# B&R Automation Studio project TD52 (part 21)

#### resetCyclic.st
```iecst
(*******************************************************************************
reset			general reset alarms
				definition remote reset capability for each individual alarm (according TI 1100-0111)

This code is confidential and proprietary to the INNIO Company.
It may not be used in any form, or reproduced in any manner,
without written permission of the INNIO Company.
Copyright, INNIO Company, 2023

Customized modifications: -
------------------------

History:
-------
V0.1	19-06-2009	Brindlinger, new
V3.10.0	12.01.2010	lettenb.	corr.for version 3.10.0
		15.02.2010	lettenb.	DO_W_QUITT, DO_A_QUITT added from task: pb8
		02.03.2010	lettenb.	extended remote reset command with T_FQUITT (was M_FQUITT)
								(needed for reset exhaust temp.alarms generated from task: exhaust)
V3.20.0	24.03.2010	lettenb.	amm numbers br9 (2201-2300) added
		21.05.2010				reset_alarm[1022,1056]: QUITT2_RUHE added
		27.05.2010				AMM test mode added, dianeblau software parts removed
		14.10.2010				NumAmmTest limited, loops reduced to 3999
V3.99.0	06.03.2013	lettenb.	adaption for pilot engine 6
								AB2MM.bResetRiskClass. added
V4.00.0 04.06.2014	lettenb.	write on VIS2MM.iNumAlarmTest removed(asynchr.running VIS do not change input field value!)
								(in case of illegal alarm nr.: alarm nr will NOT be changed, timer will NOT be started/=diff.to XT3)
		17.06.2014	lettenb.	iNumAlarmTestRun: set to 0 after alarmtest
V4.00.1 04.06.2014	lettenb.	bRemResMem: logic corr., rem.reset counter(5 resets)
V4.00.2 16.02.2015				warm-/cold restart message generation moved to MsgAB
V4.03.0 16.02.2015				protection test (gridcode III) schutzprüfung added
V4.04.0 03.11.2016				IN_AB.bResetRemBus added, prepared for future(wasserer-rosenheim)
		16.11.2016				bResetTrip: xTP_RemResCmd.Q removed, bugfix(reset all risk classes)
V4.05.1 07.03.2018	lettenb.	xR_TRIG_Run: bRun -> IN_AB.tPB2MM.bSys_Run, to avoid 1056 at PLC startup, bugfix
		21.03.2018				protection test mode: passlevel 30->15, request thaler
V4.07.1	24.06.2019	Schmid		valid alarm number space for alarm test/bypass increased from 3999 to 9999
V4.08.0	24.10.2019	Schmid		test bit for dry test bench added
V4.13.0	04.12.2023	Bencze		Risk Class 10 for remote reset of safety trips
		13.12.2023	Perktold	added A2374 as safety trip without remote reset
V4.14.0	16.12.2024	Maran		bugfix: reset of temporary alarm bypass when the Service button is switched off from HMI (issue #1621)

Instructions for use:
--------------------

Outstandings:
------------
*******************************************************************************)
PROGRAM _CYCLIC

	(*-----------------------------------------------------------------------------------------*)
	bResetLocVis			:=	VIS2MM.bResetLocVis;			(* local  reset from VIS  *)(* vis-button: 0>1 in moment of button release! *)
	bResetRemVis			:=	VIS2MM.bResetRemVis;			(* remote reset from VIS  *)(* vis-button: 0>1 in moment of button release! *)
	xF_TRIG_ResetRemExt(CLK	:=  IN_AB.tResetRemoteExt.Di		(* remote reset from DI   *)(* falling trigger according TÜV requirement *)
						    OR  IN_AB.bResetRemBus);			(* remote reset from fieldbus *)
	bResetRemExt			:=	xF_TRIG_ResetRemExt.Q;			(* falling trigger according TÜV requirement *)

	IF VIS2MM.bResetLocVis THEN VIS2MM.bResetLocVis := FALSE; END_IF;	(* reset vis data point  *)
	IF VIS2MM.bResetRemVis THEN VIS2MM.bResetRemVis := FALSE; END_IF;	(* reset vis data point *)

	(*-----------------------------------------------------------------------------------------*)
	QUITT		:=	bResetLocVis;								(* local  reset from VIS  *)
	VIS_FQUITT	:=	bResetRemVis;								(* remote reset from VIS *)
	E_FQUITT	:=	bResetRemExt;								(* remote reset from DI  *)

	(* remote reset ---------------------------------------------------------------------------*)
	bRemResIn	:= (E_FQUITT 	AND Para.bResetRemActive)		(* remote reset from DI  *)
				OR (VIS_FQUITT	AND Para.bResetRemActive);		(* remote reset from VIS *)

	(********************************************************************************************************************
	Safety-related application software source code (EN 13849-1 / 4.6.3): BEGIN
	*********************************************************************************************************************)

	(* If one of these alarms is ON, Remote Reset is deactivated *)
	IF OUT_AB.iMsg[1017]>0 OR		(* A1017 oil pressure low *)
		OUT_AB.iMsg[1019]>0 OR		(* A1019 engine cooling water pressure low *)
		OUT_AB.iMsg[1022]>0 OR		(* A1022 overspeed (relay) *)
		OUT_AB.iMsg[1026]>0 OR		(* A1026 shutdown failure *)
		OUT_AB.iMsg[1038]>0 OR		(* A1038 Generator reverse power *)
		OUT_AB.iMsg[1047]>0 OR		(* A1047: Misfiring failure *)
		(xEngType.Type6 AND OUT_AB.iMsg[1048]>0) OR		(* A1048 Knocking failure KLS90 *)
		OUT_AB.iMsg[1092]>0 OR		(* A1092 exhaust gas scavenging valve failure *)
		OUT_AB.iMsg[1131]>0 OR		(*  prepared spare - risk class 10 and this is only for trips 1,2 or 3. Remote reset is deactivated *)
		OUT_AB.iMsg[2295]>0 OR		(* A2295 engine room ventilation failure inlet air *)
		OUT_AB.iMsg[2296]>0 OR		(* A2296 engine room ventilation failure outlet air *)
		OUT_AB.iMsg[2315]>0 OR		(* A2315 air temperature before exhaust gas scavening valve maximum *)
		OUT_AB.iMsg[2337]>0 OR		(* A2337 temperature high exhaust gas pressure relief valve 1 *)
		OUT_AB.iMsg[2338]>0 OR		(* A2338 temperature high exhaust gas pressure relief valve 2 *)
		OUT_AB.iMsg[2374]>0	OR		(* A2374 Bursting disc triggered *)
		OUT_AB.iMsg[3330]>0 OR 		(* A3330 SAFI hardware failure *)
		OUT_AB.iMsg[3336]>0	OR		(* A3336 SAFI trigger signal missing *)
		OUT_AB.iMsg[3337]>0 OR		(* A3337 SAFI CAM / RESET pickup signal missing *)
		(xEngType.Type6 AND OUT_AB.iMsg[3339]>0) OR		(* A3339 Knocking failure *)
		(xEngType.Type6 AND OUT_AB.iMsg[3342]>0) OR		(* A3342 Knock sensor measuring sensor failure *)
		OUT_AB.iMsg[3343]>0 OR		(* A3343 ignition hardware failure *)
		OUT_AB.iMsg[3366]>0			(* A3366 exhaust gas scavenging fan failure *)
	THEN
		bRemResIn := FALSE;
                bRemResWarning := TRUE;
	END_IF;

	(********************************************************************************************************************
	Safety-related application software source code (EN 13849-1 / 4.6.3): END
	*********************************************************************************************************************)

	bRemResMem	:=	bRemResIn									(* remote reset memory,  unlock after: *)
				OR (bRemResMem 	AND NOT ton_FQ_timeout.Q		(* 6 h             					or *)
								AND NOT ton_oper.Q 				(* 1 h operation with closed GCB 	or *)
								AND(NOT bResetWarning OR bOMSS_MAT));(* local reset					       *)

	ton_oper(IN:= bRemResMem AND IN_AB.tGCB_On.Di AND IN_AB.tEng_Run.Do, PT:= T#1h);	(* reset after 1h load operation *)
	ton_FQ_timeout(IN:= bRemResMem, PT:=T#6h);											(* reset after 6h *)

	xR_TRIG_CD(CLK:=     bRemResIn);
	xR_TRIG_LD(CLK:= NOT bRemResMem);

	xTP_RemResCmd(IN:=  bRemResIn AND NOT xCTD_RRC.Q, PT:= T#1s);
	bRemResCmd := xTP_RemResCmd.Q;								(* remote reset command *)

	xCTD_RRC(CD:= xR_TRIG_CD.Q, LOAD:= xR_TRIG_LD.Q, PV:= 5);	(* count 5 avail.remote reset commands within 6h *)

	IF xCTD_RRC.CV=0 THEN	bRemResWarning := TRUE;				(* reached the available 5 remote reset within 1h/6h *)
	END_IF;
	(* if remote reset risk class lower than 0, the risk level is limited to 0 *)
	(* if remote reset risk class higher than 4, the risk level is limited to 4 *)
	IF Para.iResetRemRiskClass < 0 THEN Para.iResetRemRiskClass := 0;
	ELSIF Para.iResetRemRiskClass > 4 THEN Para.iResetRemRiskClass := 4;
	END_IF;

	(*-----------------------------------------------------------------------------------------*)
	xTP_Reset(IN:= QUITT OR E_QUITT, PT:= T#100ms);
	IF bDryTB_AB THEN
		xTP_DryTB_AB(IN:= bDryTB_AB, PT:= T#8h);
	ELSE
		xTP_DryTB_AB(IN:= FALSE, PT:= T#0s);
	END_IF;

	bResetWarning	:=	xTP_Reset.Q;
	bResetTrip		:=	bResetWarning AND (NOT bOMSS_MAT OR xTP_DryTB_AB.Q);

	(* remote reset commands *)
	CASE Para.iResetRemRiskClass OF
		0:	bResetRiskClass0 :=	bRemResCmd;
		1:	bResetRiskClass1 :=	bRemResCmd;
		2:	bResetRiskClass2 :=	bRemResCmd;
		3:	bResetRiskClass3 :=	bRemResCmd;
		4:	bResetRiskClass4 :=	bRemResCmd;
	END_CASE;

	(*-----------------------------------------------------------------------------------------*)
	(* monitoring on pulse (safety loop) *)
                                                        (* falling trigger according TÜV requirement *)
	xR_TRIG_Run(CLK:= IN_AB.tPB2MM.bSys_Run);			(* EN ISO 13849-1 / 5.2.2, = reset after push button release) *)
	xTP_MonOn(IN:= (xR_TRIG_Run.Q AND     IN_AB.tGCB_RUC.Do)
			    OR (QUITT         AND NOT IN_AB.tSafetyLoop_Eng.Di AND NOT bN_EngStart AND (NOT bOMSS_MAT OR xTP_DryTB_AB.Q)), PT:= T#1s);

	OUT_AB.tMonitoringOn.Do := xTP_MonOn.Q;				(* ex UW_EIN *)

	f_trig_UW_EIN(CLK:= xTP_MonOn.Q);					(* 2nd reset for safety loop *)
	QUITT2_RUHE	:= f_trig_UW_EIN.Q;
	(*-----------------------------------------------------------------------------------------*)

	IF bResetTrip OR QUITT2_RUHE THEN
		bGnlTrip1  := FALSE;
		bGnlTrip2  := FALSE;
		bGnlTrip3  := FALSE;

		bTriptype1 := FALSE;
		bTriptype2 := FALSE;
		bTriptype3 := FALSE;
	END_IF;

	IF bResetWarning THEN
		bGnlWarning := FALSE;
		bRemResWarning := FALSE;
	END_IF;

	(*-----------------------------------------------------------------------------------------*)
	xTP_ResetWarning(IN:= bResetWarning, PT:= T#1s);		(* DO's for acknowledgement *)
	OUT_AB.tResetWarning.Do := xTP_ResetWarning.Q;

	xTP_ResetTrip(IN:= bResetTrip, PT:= T#1s);
	OUT_AB.tResetTrip.Do    := xTP_ResetTrip.Q;

	(*-----------------------------------------------------------------------------------------*)
	(* ----------------------------------------------------------------------------------------*)
	(* AMM test mode *)
	//	in:		iNumAlarmTest	bAlarmTestStart		bAlarmTestStop
	//			iPassLevel		bServiceBegin
	//	out:	bAlarmTestOn	bAlarmTestEnable	iAlarmTestRestTime	[in s]

	(* service mode on/off *)
	xTON_ServiceTimeOut(IN:= (IN_AB.tGCB_On.Di AND VIS2MM.bServiceBegin), PT:= T#2h);	(* reset timer - after 2 hours with closed gen-c.b. reset service button *)

	IF xTON_ServiceTimeOut.Q THEN
		VIS2MM.bServiceBegin := FALSE;			(* reset timer from ctr *)
	ELSE
		VIS2MM.bServiceBegin;					(* set/reset timer from vis *)
	END_IF;

	OUT_AB.bServiceMode := VIS2MM.bServiceBegin;

	(*-----------------------------------------------------------------------------------*)
	VIS2MM.bAlarmTestStart;
	iNumAlarmTest	:= VIS2MM.iNumAlarmTest;//LIMIT(VIS2MM.iNumAlarmTest,1001,3999);
	VIS2MM.bAlarmTestStop;

	IF OUT_AB.bServiceMode AND IN_AB.iPassLevel >= 30 THEN
		bAlarmTestEnable := TRUE;
		(*-----------------------------------------------------------------------------------*)
		IF Para.bVISA THEN
			CASE iNumAlarmTest OF
				1021:	iNumAlarmTest := 0;
				1023:	iNumAlarmTest := 0;
				1028:	iNumAlarmTest := 0;
				1030:	iNumAlarmTest := 0;
				1135:	iNumAlarmTest := 0;
				1057:	iNumAlarmTest := 0;
				1058:	iNumAlarmTest := 0;
			END_CASE;
		END_IF;

		CASE iNumAlarmTest OF
			1022:	iNumAlarmTest := 0;
			1026:	iNumAlarmTest := 0;
			1031:	iNumAlarmTest := 0;
			1033:	iNumAlarmTest := 0;
			1034:	iNumAlarmTest := 0;
			1035:	iNumAlarmTest := 0;
			1038:	iNumAlarmTest := 0;
			1041:	iNumAlarmTest := 0;
			1042:	iNumAlarmTest := 0;
			1053:	iNumAlarmTest := 0;
			1054:	iNumAlarmTest := 0;
			1056:	iNumAlarmTest := 0;	(* ruhestromschleife unterbrochen	*)
			1061:	iNumAlarmTest := 0;	(* zündung gestört					*)
			3025:	iNumAlarmTest := 0;
			3026:	iNumAlarmTest := 0;
			3027:	iNumAlarmTest := 0;
			3028:	iNumAlarmTest := 0;
			3029:	iNumAlarmTest := 0;
			3310:	iNumAlarmTest := 0;
			3330:	iNumAlarmTest := 0;
			3333:	iNumAlarmTest := 0;
			3335:	iNumAlarmTest := 0;
			3336:	iNumAlarmTest := 0;
			3337:	iNumAlarmTest := 0;
			3344:	iNumAlarmTest := 0;
			3345:	iNumAlarmTest := 0;
		END_CASE;

		IF    iNumAlarmTest < 1001 THEN iNumAlarmTest := 0;
		ELSIF iNumAlarmTest > 9999 THEN iNumAlarmTest := 0;
		END_IF;

		IF    iNumAlarmTest <> 0   THEN NumAmmTestValid := TRUE;
		ELSE					        NumAmmTestValid := FALSE;
		END_IF;

		(*-----------------------------------------------------------------------------------*)
		(* start alarm test from visu-button *)
		r_trig_SetAmmTestStart(CLK:= VIS2MM.bAlarmTestStart AND NumAmmTestValid);
		IF r_trig_SetAmmTestStart.Q THEN
			tp_AmmTestReset(IN:= FALSE, PT:=T#0s);
			tp_AmmTestReset.IN:= VIS2MM.bAlarmTestStart;
			tp_AmmTestReset.PT:= T#300s;
			iNumAlarmTestX    := iNumAlarmTest;
		END_IF;
		VIS2MM.bAlarmTestStart := FALSE;	(* reset vis datapoint *)

		tp_AmmTestReset();

		IF VIS2MM.bAlarmTestStop THEN
			tp_AmmTestReset(IN:= FALSE, PT:=T#0s);
		END_IF;
		VIS2MM.bAlarmTestStop := FALSE;		(* reset vis datapoint *)

		bAlarmTestOn			:= tp_AmmTestReset.Q;

		(* alarm test rest time for visu *)
		IF bAlarmTestOn THEN
			iNumAlarmTest      	:= iNumAlarmTestX;
			iNumAlarmTestRun	:= iNumAlarmTestX;		(* number alarm test running > meta modules *)
			iAlarmTestRestTime	:= DINT_TO_INT(TIME_TO_DINT(tp_AmmTestReset.PT - tp_AmmTestReset.ET)/1000);
		ELSE
			iNumAlarmTestRun   	:= 0;
			iAlarmTestRestTime	:= 0;
		END_IF;

	ELSE
		VIS2MM.bAlarmTestStart	:= FALSE;
		VIS2MM.bAlarmTestStop	:= FALSE;
		bAlarmTestEnable 		:= FALSE;
		bAlarmTestOn			:= FALSE;
		iNumAlarmTest			:= 0;
		iNumAlarmTestRun		:= 0;
		iAlarmTestRestTime		:= 0;
		tp_AmmTestReset(IN:= FALSE, PT:=T#0s);
	END_IF;

	MM2VIS.bNumAmmTestValid := NumAmmTestValid;

	(*-----------------------------------------------------------------------------------*)
	(* protection test (gridcode III) schutzprüfung -------------------------------------*)
	VIS2MM.bMMD_GenAlarmTestStart;		VIS2MM.bMMD_GenAlarmTestStop;
	VIS2MM.bMMD_BB_AlarmTestStart;		VIS2MM.bMMD_BB_AlarmTestStop;

	(* protection test mode on/off *)
	IF 		 	IN_AB.iPassLevel >= 15
		AND 	bOMSS_Stop
		AND 	xOpMode.Stop	THEN	bMMD_GenAlarmTestEnable := TRUE;
										bMMD_BB_AlarmTestEnable := TRUE;

		(*-----------------------------------------------------------------------------------*)
		(* start GenAlarmTest from visu-button *)
		r_trig_SetMMD_GenAmmTestStart(CLK:= VIS2MM.bMMD_GenAlarmTestStart AND bMMD_GenAlarmTestEnable);
		IF r_trig_SetMMD_GenAmmTestStart.Q THEN
			tp_MMD_GenAmmTestReset(IN:= FALSE, PT:=T#0s);
			tp_MMD_GenAmmTestReset.IN:= VIS2MM.bMMD_GenAlarmTestStart;
			tp_MMD_GenAmmTestReset.PT:= T#30m;
		END_IF;
		VIS2MM.bMMD_GenAlarmTestStart := FALSE;	(* reset vis datapoint *)

		tp_MMD_GenAmmTestReset();

		IF VIS2MM.bMMD_GenAlarmTestStop THEN
			tp_MMD_GenAmmTestReset(IN:= FALSE, PT:=T#0s);
		END_IF;
		VIS2MM.bMMD_GenAlarmTestStop := FALSE;		(* reset vis datapoint *)

		bMMD_GenAlarmTestOn		:= tp_MMD_GenAmmTestReset.Q;

		(* alarm test rest time for visu *)
		IF bMMD_GenAlarmTestOn THEN
			iMMD_GenAlarmTestRestTime	:= DINT_TO_INT(TIME_TO_DINT(tp_MMD_GenAmmTestReset.PT - tp_MMD_GenAmmTestReset.ET)/1000);
		ELSE
			iMMD_GenAlarmTestRestTime	:= 0;
		END_IF;

		(*-----------------------------------------------------------------------------------*)
		(* start BB_AlarmTest from visu-button *)
		r_trig_SetMMD_BB_AmmTestStart(CLK:= VIS2MM.bMMD_BB_AlarmTestStart AND bMMD_BB_AlarmTestEnable);
		IF r_trig_SetMMD_BB_AmmTestStart.Q THEN
			tp_MMD_BB_AmmTestReset(IN:= FALSE, PT:=T#0s);
			tp_MMD_BB_AmmTestReset.IN:= VIS2MM.bMMD_BB_AlarmTestStart;
			tp_MMD_BB_AmmTestReset.PT:= T#30m;
		END_IF;
		VIS2MM.bMMD_BB_AlarmTestStart := FALSE;	(* reset vis datapoint *)

		tp_MMD_BB_AmmTestReset();

		IF VIS2MM.bMMD_BB_AlarmTestStop THEN
			tp_MMD_BB_AmmTestReset(IN:= FALSE, PT:=T#0s);
		END_IF;
		VIS2MM.bMMD_BB_AlarmTestStop := FALSE;		(* reset vis datapoint *)

		bMMD_BB_AlarmTestOn		:= tp_MMD_BB_AmmTestReset.Q;

		(* BB_AlarmTest rest time for visu *)
		IF bMMD_BB_AlarmTestOn THEN
			iMMD_BB_AlarmTestRestTime	:= DINT_TO_INT(TIME_TO_DINT(tp_MMD_BB_AmmTestReset.PT - tp_MMD_BB_AmmTestReset.ET)/1000);
		ELSE
			iMMD_BB_AlarmTestRestTime	:= 0;
		END_IF;

	ELSE
		VIS2MM.bMMD_GenAlarmTestStart	:= FALSE;
		VIS2MM.bMMD_GenAlarmTestStop	:= FALSE;
		bMMD_GenAlarmTestEnable 		:= FALSE;
		bMMD_GenAlarmTestOn				:= FALSE;
		tp_MMD_GenAmmTestReset(IN:= FALSE, PT:=T#0s);
		iMMD_GenAlarmTestRestTime		:= 0;

		VIS2MM.bMMD_BB_AlarmTestStart	:= FALSE;
		VIS2MM.bMMD_BB_AlarmTestStop	:= FALSE;
		bMMD_BB_AlarmTestEnable 		:= FALSE;
		bMMD_BB_AlarmTestOn				:= FALSE;
		tp_MMD_BB_AmmTestReset(IN:= FALSE, PT:=T#0s);
		iMMD_BB_AlarmTestRestTime		:= 0;
	END_IF;

	OUT_AB.bMMD_GenAlarmTestOn := bMMD_GenAlarmTestOn;
	OUT_AB.bMMD_BB_AlarmTestOn := bMMD_BB_AlarmTestOn;
	(*-----------------------------------------------------------------------------------*)
END_PROGRAM
```

#### resetInit.st
```iecst
(*******************************************************************************
reset			general reset alarms
				definition remote reset capability for each individual alarm (according TI 1100-0111)

This code is confidential and proprietary to the INNIO Company.
It may not be used in any form, or reproduced in any manner,
without written permission of the INNIO Company.
Copyright, INNIO Company, 2019

Customized modifications: -
------------------------

History:
-------
V0.1	19-06-2009	Brindlinger, new
V3.10.0	12.01.2010	lettenb.	corr.for version 3.10.0
		15.02.2010	lettenb.	DO_W_QUITT, DO_A_QUITT added from task: pb8
		02.03.2010	lettenb.	extended remote reset command with T_FQUITT (was M_FQUITT)
								(needed for reset exhaust temp.alarms generated from task: exhaust)
V3.20.0	24.03.2010	lettenb.	amm numbers br9 (2201-2300) added
		21.05.2010				reset_alarm[1022,1056]: QUITT2_RUHE added
		27.05.2010				AMM test mode added, dianeblau software parts removed
		14.10.2010				NumAmmTest limited, loops reduced to 3999
V3.99.0	06.03.2013	lettenb.	adaption for pilot engine 6
								AB2MM.bResetRiskClass. added
V4.00.0 04.06.2014	lettenb.	write on VIS2MM.iNumAlarmTest removed(asynchr.running VIS do not change input field value!)
								(in case of illegal alarm nr.: alarm nr will NOT be changed, timer will NOT be started/=diff.to XT3)
		17.06.2014	lettenb.	iNumAlarmTestRun: set to 0 after alarmtest
V4.00.1 04.06.2014	lettenb.	bRemResMem: logic corr., rem.reset counter(5 resets)
V4.00.2 16.02.2015				warm-/cold restart message generation moved to MsgAB
V4.03.0 16.02.2015				protection test (gridcode III) schutzprüfung added
V4.04.0 03.11.2016				IN_AB.bResetRemBus added, prepared for future(wasserer-rosenheim)
		16.11.2016				bResetTrip: xTP_RemResCmd.Q removed, bugfix(reset all risk classes)
V4.05.1 07.03.2018	lettenb.	xR_TRIG_Run: bRun -> IN_AB.tPB2MM.bSys_Run, to avoid 1056 at PLC startup, bugfix
		21.03.2018				protection test mode: passlevel 30->15, request thaler
V4.07.1	24.06.2019	Schmid		valid alarm number space for alarm test/bypass increased from 3999 to 9999
V4.08.0	24.10.2019	Schmid		test bit for dry test bench added

Instructions for use:
--------------------

Outstandings:
------------
*******************************************************************************)
PROGRAM _INIT

	(* Reset Dry TB variable *)
	 bDryTB_AB := FALSE;

END_PROGRAM
```

#### reset.var
```iecst
VAR
	bResetRemVis : BOOL;
	bResetLocVis : BOOL;
	bResetRemExt : BOOL;
	iNumAlarmTestX : DINT; (*number alarm test*)
	iNumAlarmTest : DINT; (*number alarm test*)
	QUITT : BOOL;
	VIS_FQUITT : BOOL;
	r_trig_SetAmmTestStart : R_TRIG := (0);
	f_trig_UW_EIN : F_TRIG := (0);
	ton_FQ_timeout : TON := (0);
	xR_TRIG_CD : R_TRIG := (0);
	xR_TRIG_LD : R_TRIG := (0);
	xCTD_RRC : CTD := (0);
	ton_oper : TON := (0);
	NumAmmTestValid : BOOL := FALSE;
	tp_AmmTestReset : TP := (0);
	E_FQUITT : BOOL;
	QUITT2_RUHE : BOOL;
	xR_TRIG_Run : R_TRIG := (0);
	xTP_MonOn : TP := (0);
	bRemResMem : BOOL;
	E_QUITT : BOOL;
	xTP_RemResCmd : TP;
	xTP_ResetWarning : TP;
	xTP_ResetTrip : TP;
	xTP_Reset : TP;
	xF_TRIG_ResetRemExt : F_TRIG;
	xTON_ServiceTimeOut : TON;
	tp_MMD_GenAmmTestReset : TP := (0);
	r_trig_SetMMD_GenAmmTestStart : R_TRIG := (0);
	tp_MMD_BB_AmmTestReset : TP := (0);
	r_trig_SetMMD_BB_AmmTestStart : R_TRIG := (0);
	bDryTB_AB : BOOL;
	xTP_DryTB_AB : TP;
END_VAR
```

### Program Logical/AmmBase/AmmGnl (IEC) - + alarm management general

- AmmGnlCyclic.st (not readable text: treated as protected, skipped)

#### AmmGnl.var
```iecst
VAR
	xTON_StopM : TON;
END_VAR
```

### Program Logical/AmmBase/MsgAB (IEC, version 4.13.0) - message

#### MsgABCyclic.st
```iecst
(*******************************************************************************
MsgAB	 			 alarms generation

This code is confidential and proprietary to the INNIO Company.
It may not be used in any form, or reproduced in any manner,
without written permission of the INNIO Company.
Copyright, INNIO Company, 2023

Customized modifications: -
------------------------

History:
-------
V0.01.0	02.11.2011	lettenb.	new
V3.99.0	07.03.2013	lettenb.	cleanup
		24.05.2013				reset OUT_xx.txx2AB.bGnlTripx changed
		07.11.2013				bMsg3003 removed, cleanup
V4.00.0	27.02.2014				logger added
V4.00.1	17.12.2014				3003 modif.for 920(920 stapelfeld), enable with IN_AB.tPB2MM.bSys_Run
V4.04.0	21.10.2016	lettenb.	3003(2103,2104) modif.for functional safety(thummer/feyrsinger/gföller)
		28.07.2017	502423184	no shut down due TO a measuring signal failure, SWAT #3
V4.05.0	22.12.2017	lettenb.	comment added: Safety-related application software source code (EN 13849-1 / 4.6.3)#
		22.01.2018	lettenb.	3003 bSys_Run -> bParaSetupOk to avoid message at plc startup
V4.13.0	04.12.2023	Bencze		Risk Class 10 for remote reset of safety trips
V4.14.0 06.11.2024 Nagy bMsg3152 Room Temperature Signal Failure removed from A3003 2024-226 Trip Desent

Instructions for use:
--------------------
1) declare alarm with function block "Msg"
	declare buffert alarm bit bMsg<message number>

2) use template to create a new alarm,
   substitue 0000 by alarm number and make settings:

	xMsg0000.Enable		:=	TRUE;		enable/disable alarm
	xMsg0000.Set		:=	FALSE;		alarm set condition
	xMsg0000.PT			:=	T#0s;		alarm delay time
	xMsg0000.Prio		:=	1;			alarm priority: 1-3 = trip, 4 = warning
	xMsg0000.RiskClass	:=	3;			risk class for remote alarm reset acc.TI 1100-0111
	xMsg0000.Reset		:=	FALSE;		FALSE: for all standard alarms	prio 1,2,3 and warnings prio 4
										TRUE : for autoreset alarms

	bMsg0000			:=	xMsg0000.Q;	connect buffert alarm bit for VIS and control
	bMsg0000_Test		:=	xMsg0000.Test; alarm bypass active

3)  expand INIT

Outstandings:
------------
(*******************************************************************************)
PROGRAM _CYCLIC

	(* reset general trip *)
	tMM2AB.bGnlTrip1	:=	FALSE;
	tMM2AB.bGnlTrip2	:=	FALSE;
	tMM2AB.bGnlTrip3	:=	FALSE;
	tMM2AB.bGnlWarning	:=	FALSE;
	tMM2AB.bTriptype1	:=	FALSE;
	tMM2AB.bTriptype2	:=	FALSE;
	tMM2AB.bTriptype3	:=	FALSE;

	(********************************************************************************************************************
	Safety-related application software source code (EN 13849-1 / 4.6.3): BEGIN
	*********************************************************************************************************************)
	(* W3003 signal failure( 2101 or 2102 or 2103 or 2104 *)
	xMsg3003.Enable	   := IN_AB.tPB2MM.bParaSetupOk;
	IF xEngType.Type9 THEN

		xMsg3003.Set   :=   IN_AB.bMsg2101
						OR  IN_AB.bMsg2102
	//					OR  IN_AB.bMsg2103		(* no shut down due to a measuring signal failure, SWAT #3 *)
						OR  IN_AB.bMsg2104;
	ELSE
		bSigFail	   :=	IN_AB.bMsg2101 OR IN_AB.bMsg2102;
		xTON_SigFail(IN:= bSigFail, PT:= T#24h);
		xTON_SigFail_2103(IN:= IN_AB.bMsg2103, PT:= T#30s);
		xTON_SigFail_2104(IN:= IN_AB.bMsg2104, PT:= T#30s);

		xMsg3003.Set   :=  (bSigFail OR IN_AB.bMsg2103 OR IN_AB.bMsg2104)
				AND(	    xTON_SigFail.Q
					OR		xTON_SigFail_2103.Q
					OR		xTON_SigFail_2104.Q
					OR  NOT IN_AB.tEng_Run.Do
					OR(    (IN_AB.bMsg2101 OR IN_AB.bMsg2104) AND(IN_AB.bMsg2102 OR IN_AB.bMsg2103))
					OR		xMsg3003.Set);
	END_IF;
	xMsg3003.PT	       := T#0s;
	xMsg3003.Prio 	   := 3;
	xMsg3003.RiskClass := 4;
	xMsg3003.Reset 	   := TRUE;		(* autoreset *)
	xMsg3003();
	OUT_AB.bMsg3003    := xMsg3003.Q;
	MM2VIS.bMsg3003    := xMsg3003.Q;
	(********************************************************************************************************************
	Safety-related application software source code (EN 13849-1 / 4.6.3): END
	*********************************************************************************************************************)

	(*---------------------------------------------------------------------------*)
	(* operating messages *)

	(* B1239 general trip *)
	xMsg1239.Enable		:=	IN_AB.tPB2MM.bSys_Run;
	xMsg1239.Set		:=	bGnlTrip;
	xMsg1239.Reset		:=	TRUE;
	xMsg1239();
	MM2VIS.bMsg1239		:= xMsg1239.Q;

	(* B1240 general warning *)
	xTOF_GnlWarning(IN:= bGnlWarning, PT:= T#1s); (* to avoid message with resistent bGnlWarning *)

	xMsg1240.Enable		:=	IN_AB.tPB2MM.bSys_Run;
	xMsg1240.Set		:=	xTOF_GnlWarning.Q;
	xMsg1240.Reset		:=	TRUE;
	xMsg1240();
	MM2VIS.bMsg1240		:= xMsg1240.Q;

	(* B1253 warm restart *)
	xTOF_WarmRestart(IN:= NOT bWarmRestart, PT:= T#3m);
	bWarmRestart := TRUE;

	xMsg1253.Enable		:=	FALSE;	(* no permanent memory available *)
	xMsg1253.Set		:=	xTOF_WarmRestart.Q;
	xMsg1253.Reset		:=	TRUE;
	xMsg1253();
	MM2VIS.bMsg1253		:= xMsg1253.Q;

	(* B1254 cold restart *)
	xTOF_ColdRestart(IN:= NOT bColdRestart, PT:= T#3m);
	bColdRestart := TRUE;

	xMsg1254.Enable		:=	TRUE;
	xMsg1254.Set		:=	xTOF_ColdRestart.Q;
	xMsg1254.Reset		:=	TRUE;
	xMsg1254();
	MM2VIS.bMsg1254		:= xMsg1254.Q;

	(* B1256 reset *)
	xMsg1256.Enable		:=	TRUE;
	xMsg1256.Set		:=	bResetWarning;
	xMsg1256.Reset		:=	TRUE;
	xMsg1256();
	MM2VIS.bMsg1256		:= xMsg1256.Q;

	(* B3252 remote reset *)
	xMsg3252.Enable		:=	TRUE;
	xMsg3252.Set		:=	bRemResCmd;
	xMsg3252.Reset		:=	TRUE;
	xMsg3252();
	MM2VIS.bMsg3252		:= xMsg3252.Q;

	(* W9389 Remote acknowledgement not possible (too many or safety trip) *)
	xMsg9389.Enable		:= Para.iResetRemRiskClass > 0;
	xMsg9389.Set		:= bRemResWarning;
	xMsg9389.PT	        := T#0s;
	xMsg9389.Prio 	    := 4;
	xMsg9389.RiskClass  := 4;
	xMsg9389();
	MM2VIS.bMsg9389		:= xMsg9389.Q;

	(* B template
	xMsg.Enable		:=	TRUE;
	xMsg.Set		:=	bBool;
	xMsg.Reset		:=	TRUE;
	xMsg();
	MM2VIS.bMsg		:= xMsg.Q;
	*)

	(*---------------------------------------------------------------------------*)
	(* general alarms for further module operations *)
	bGnlTrip1_AB	:= tAB2MM.bGnlTrip1   OR tMM2AB.bGnlTrip1;
	bGnlTrip2_AB	:= tAB2MM.bGnlTrip2   OR tMM2AB.bGnlTrip2;
	bGnlTrip3_AB	:= tAB2MM.bGnlTrip3   OR tMM2AB.bGnlTrip3;
	bGnlWarning_AB	:= tAB2MM.bGnlWarning OR tMM2AB.bGnlWarning;

	bGnlTrip_AB		:= bGnlTrip1_AB OR bGnlTrip2_AB OR bGnlTrip3_AB;

(*******************************************************************************)
END_PROGRAM
```

#### MsgABInit.st
```iecst
(*******************************************************************************
Msg_AB	 			 alarms generation

This code is confidential and proprietary to the INNIO Company.
It may not be used in any form, or reproduced in any manner,
without written permission of the INNIO Company.
Copyright, INNIO Company, 2023

Customized modifications: -
------------------------

History:
-------
V0.00.0	29.07.2011	lettenb.	new
V3.99.0	07.03.2013	lettenb.	cleanup
V4.13.0	04.12.2023	Bencze		Risk Class 10 for remote reset of safety trips

Instructions for use:
--------------------
1) declare alarm with function block "Msg"

2) use template to create a new alarm, substitue 0000 by message number:

	xMsg0000.Num		:=	0000;					alarm number
	xMsg0000.AmmSysAdr	:=  iAdrAmmBase2MM;			do not change
	xMsg0000.AmmOutAdr	:=  iAdrMM2AmmBase;			do not change

3) 	set alarm number

Outstandings:
------------
(*******************************************************************************)
PROGRAM _INIT

	iAdrAmmBase2MM		:=  ADR(tAB2MM);//ADR(OUT_AB.tAB2MM);
	iAdrMM2AmmBase		:=  ADR(tMM2AB);//ADR(IN_AB.tMM2AB);

	(*---------------------------------------------------------------------------*)

	xMsg1239.Num		:=	1239;
	xMsg1239.AmmInAdr	:=  iAdrAmmBase2MM;
	xMsg1239.AmmOutAdr	:=  iAdrMM2AmmBase;

	xMsg1240.Num		:=	1240;
	xMsg1240.AmmInAdr	:=  iAdrAmmBase2MM;
	xMsg1240.AmmOutAdr	:=  iAdrMM2AmmBase;

	xMsg1253.Num		:=	1253;
	xMsg1253.AmmInAdr	:=  iAdrAmmBase2MM;
	xMsg1253.AmmOutAdr	:=  iAdrMM2AmmBase;

	xMsg1254.Num		:=	1254;
	xMsg1254.AmmInAdr	:=  iAdrAmmBase2MM;
	xMsg1254.AmmOutAdr	:=  iAdrMM2AmmBase;

	xMsg1256.Num		:=	1256;
	xMsg1256.AmmInAdr	:=  iAdrAmmBase2MM;
	xMsg1256.AmmOutAdr	:=  iAdrMM2AmmBase;

	xMsg3252.Num		:=	3252;
	xMsg3252.AmmInAdr	:=  iAdrAmmBase2MM;
	xMsg3252.AmmOutAdr	:=  iAdrMM2AmmBase;

	xMsg3003.Num		:=	3003;
	xMsg3003.AmmInAdr	:=  iAdrAmmBase2MM;
	xMsg3003.AmmOutAdr	:=  iAdrMM2AmmBase;

	(* W9389 Remote acknowledgement not possible, too many or safety trip *)
	xMsg9389.Num		:=	9389;
	xMsg9389.AmmInAdr	:=  iAdrAmmBase2MM;
	xMsg9389.AmmOutAdr	:=  iAdrMM2AmmBase;

	(* template
	xMsg.Num		:=	;
	xMsg.AmmInAdr	:=  iAdrAmmBase2MM;
	xMsg.AmmOutAdr	:=  iAdrMM2AmmBase;
	*)

END_PROGRAM
```

#### MsgAB.var
```iecst
VAR
	iAdrAmmBase2MM : UDINT;
	iAdrMM2AmmBase : UDINT;
	bSigFail : BOOL;
	xTON_SigFail : TON;
	xTON_SigFail_2103 : TON;
	xTON_SigFail_2104 : TON;
	xMsg1239 : Msg;
	xMsg1240 : Msg;
	xMsg1253 : Msg;
	xMsg1254 : Msg;
	xMsg1256 : Msg;
	xMsg3252 : Msg;
	xMsg3003 : Msg;
	xMsg9389 : Msg;	(* W9389 Remote acknowledgement not possible, too many or safety trip *)
	bGnlTrip_AB : BOOL; (*general trip - common (MM_AB local)*)
	bGnlTrip1_AB : BOOL; (*general trip priority 1 - common (MM_AB local)*)
	bGnlTrip2_AB : BOOL; (*general trip priority 2 - common (MM_AB local)*)
	bGnlTrip3_AB : BOOL; (*general trip priority 3 - common (MM_AB local)*)
	bGnlWarning_AB : BOOL; (*general warning - common (MM_AB local)*)
	xTOF_GnlWarning : TOF;
END_VAR
```

### Program Logical/AmmBase/vis_AB (IEC, version 4.09.0) - visualization

#### vis_ABCyclic.st
```iecst
(*******************************************************************************
vis			visualization

This code is confidential and proprietary to the INNIO Company.
It may not be used in any form, or reproduced in any manner,
without the express written permission of the INNIO Company.
Copyright, INNIO Company, 2020

Customized modifications: -
------------------------

History:
-------
V0.00.0	24.04.2012	lettenb.	new
V3.99.0	07.03.2013	lettenb.	cleanup
		07.11.2013				messages setted in MsgAB removed, cleanup
V4.03.0 16.02.2015				protection test (gridcode III) schutzprüfung added
V4.09.0	19.03.2020	lettenb.	protection test: bMMD_BB_AlarmTestEnable, bMMD_BB_AlarmTestOn for VIS added

Instructions for use:
--------------------
Outstandings:
------------
*******************************************************************************)
PROGRAM _CYCLIC

	MM2VIS.bGnlTrip1			:=		bGnlTrip1;
	MM2VIS.bGnlTrip2			:=		bGnlTrip2;
	MM2VIS.bGnlTrip3			:=		bGnlTrip3;
	MM2VIS.bGnlTrip				:=		bGnlTrip;
	MM2VIS.bGnlWarning			:=		bGnlWarning;

	MM2VIS.bTriptype1			:=		bTriptype1;
	MM2VIS.bTriptype2			:=		bTriptype2;
	MM2VIS.bTriptype3			:=		bTriptype3;
	MM2VIS.bTriptypeS			:=	NOT IN_AB.tSafetyLoop_Eng.Di;

	MM2VIS.bGnlTripDurEngOp;
	MM2VIS.bAlarmTestEnable		:=		bAlarmTestEnable;
	MM2VIS.bAlarmTestOn			:=		bAlarmTestOn;
	MM2VIS.iAlarmTestRestTime	:=		iAlarmTestRestTime;

	MM2VIS.bMMD_GenAlarmTestEnable		:=	bMMD_GenAlarmTestEnable;
	MM2VIS.bMMD_GenAlarmTestOn			:=	bMMD_GenAlarmTestOn;
	MM2VIS.iMMD_GenAlarmTestRestTime	:=	iMMD_GenAlarmTestRestTime;

	MM2VIS.bMMD_BB_AlarmTestEnable		:=	bMMD_BB_AlarmTestEnable;
	MM2VIS.bMMD_BB_AlarmTestOn			:=	bMMD_BB_AlarmTestOn;
	MM2VIS.iMMD_BB_AlarmTestRestTime	:=	iMMD_BB_AlarmTestRestTime;

END_PROGRAM
```

### Program Logical/AmmBase/ParAB (IEC, version 4.07.0) - + parameter handling

- perm_par.st (not readable text: treated as protected, skipped)

#### perm_par.var
```iecst
VAR
	tParaIntern : ParaHandler_typ; (*Connector type to perm_par*)
	tMM2ParaBase_ReadBack : MM2ParaBase_type; (*INTERNAL! V4.06 new readback structure for information from previous tasks*)
	bWriteDataObj : BOOL; (* TRUE=write data object module *)
	bDataObjLenErr : BOOL; (*Error occured in permem: data module size missmatch*)
	bCreateDataObj : BOOL; (* TRUE=create new data object *)
	bWriteOnce : BOOL; (* write permanent memory once *)
	DatObjCreate_01 : DatObjCreate; (* data object create *)
	DatObjInfoBak_02 : DatObjInfo; (* data object info *)
	DatObjDelete_01 : DatObjDelete; (* data object delete *)
	DatObjRead_01 : DatObjRead; (* data object read *)
	DatObjRead_02 : DatObjRead; (* manual initiated data object read *)
	DatObjWrite_01 : DatObjWrite; (* data object write *)
	DatObjDelete_02 : DatObjDelete; (* data object delete *)
	DatObjDelete_11 : DatObjDelete; (*Delete Backup File*)
	DatObjInfo_01 : DatObjInfo; (* data object info *)
	DatObjInfo_02 : DatObjInfo; (* data object info *)
	szModuleName : STRING[35]; (* module name of object *)
	szModuleNameBackup : STRING[35]; (* module name of posiibly created backup object *)
	DatObjCopy_01 : DatObjCopy;
	bCopyDataObj : BOOL;
	TON_WarnDelay : TON;
	TON_WritePMEM : TON; (* delay write permanent memory *)
	ulPMPointer : UDINT; (* adress of actual checksum value *)
	ulChecksum : UDINT; (* parameter checksum value *)
	pm_len : UDINT; (* permanent value lenght *)
	ulChecksumOld : UDINT; (* last vlaue of parameter checksum *)
	ulChkValue : UDINT; (* actual value of parameter pointer *)
	pm_id : UDINT; (* permanent value identifier *)
	pm_p : UDINT; (* permanent value pointer *)
	DatObjInfo_META : DatObjInfo;
	DatObjRead_META : DatObjRead;
	szMetaDataRaw : STRING[2000];
	szMetaData : ARRAY[0..4] OF STRING[35];
	szMetaDataVis : ARRAY[0..3] OF STRING[35];
	ssIndex : INT;
	ssCount : INT;
	ucMetaDataRaw : ARRAY[0..2000] OF USINT;
	ssCount2 : INT;
	szMetaDataFile : STRING[10];
	szText1 : STRING[20];
	pv_adr_IN_XX_tPB2MM : UDINT;
	pv_lng : UDINT;
	pv_lng_IN_XX_tPB2MM : UDINT;
	pv_lng_OUT_XX_tPB2MM : UDINT;
	szText2 : STRING[20];
	pv_adr_OUT_XX_tXX2PB : UDINT;
END_VAR
VAR CONSTANT
	ERR_NOERROR : UINT := 0;
END_VAR
VAR
	usPMWriteCnt : UINT;
	pm_Error : UDINT; (* permanent value error *) (* Deleted: pm : ParaMem_typ; permanent memory tags mathias, 22.8.11*)
	fun_Error : UDINT := 0; (*state > 0 = function error*)
	xLocalParaCheck : ParaCheckFUB; (*local function instance to check parameter values*)
	TON_ParaSetupOk : TON;
	bParaCheckSystemOk : BOOL;
	iDebug_ParaOkChecked : UDINT;
	bRestoreBackupDataObj : BOOL := FALSE;
	bRestoreDataObjContent : BOOL := FALSE;
	pm_id_backup : UDINT;
	pm_p_Backup : UDINT;
	DatObjCopy_02 : DatObjCopy;
	bDeleteBackupDataObj : BOOL := FALSE; (*Command to delete backup data module file on purpose*)
	bDebugPara : ARRAY[0..5] OF BOOL;
	ssIndex2 : INT;
	ssIndex3 : INT;
	ssIndex4 : INT;
	ssIndexVis : INT;
	szText : STRING[40];
	pv_adr_Para : UDINT;
	szParaSnippet : ARRAY[0..5] OF STRING[150];
	szParaIndex : STRING[10];
	slValue : DINT;
	iModuleDLD_ResetCount : INT;
	bDownloadDetected : BOOL;
	bFlagParaStructCopyWorking : BOOL; (*true, if cyclic para copying is active, 1 false cycle at every copy *)
	bStoreInitParaInDataObj : BOOL := FALSE;
	bTestflag : BOOL;
	bReadOutMETA_Once : BOOL;
	tParaCheck_iPvAdress : ARRAY[0..5] OF UDINT;
	tParaCheck_iPvLengt : ARRAY[0..5] OF UDINT;
	tParaCheck_rPvValue : ARRAY[0..5] OF REAL;
	tParaCheck_rRangeMIN : ARRAY[0..5] OF REAL;
	tParaCheck_rRangeMAX : ARRAY[0..5] OF REAL;
	tParaCheck_szPvName : ARRAY[0..5] OF STRING[35];
	ssFormatDetected : INT;
	szMetaDataPart : STRING[150];
	szFullTaskName : STRING[35];
	szFullMetaModuleName : STRING[35];
	debugLen : INT;
	debugSize : INT := 0;
	strcat_adr1 : UDINT;
	strcat_adr2 : UDINT;
	ssIndexTN : INT;
	bAlternate : BOOL;
	n : INT;
	iAlternateChecksum : DINT;
	iAlternateChecksumOld : DINT;
	ulDebugChkValue : ARRAY[0..999] OF UDINT;
	Adr1 : UDINT;
	Adr2 : UDINT;
	usPMWriteCntStepsize : UINT := 1; (*different step sizes to help debug*)
	usPMWriteCntXOR : UINT;
	usPMWriteCntAltSum : UINT;
	ulAdrPM : UDINT;
	usChkValuePM : USINT;
	ulAdrPara : UDINT;
	ulPara_len : UDINT;
	usChkValuePara : USINT;
	iDebugCountPMDifferences : DINT := 0;
	bEngineRunDetected : BOOL; (*detection status bit autocommand 100 /101  for engine run state*)
	ucMetaDataDebugInfoLine : ARRAY[0..24] OF STRING[80];
	ssIndexMand : INT := 0;
	szMetaDataMand : STRING[35];
	iMyErrorInfo_Autoreset : DINT; (*internal autoreset counter*)
	ssIndex_Version : INT; (*internal*)
	ssIndex_BU : INT; (*internal*)
	ssIndex_BU2 : INT; (*internal*)
END_VAR
```

### Program Logical/AmmBase/AmmGnlTC5 (IEC) - + alarm management general

- AmmGnlTC5Cyclic.st (not readable text: treated as protected, skipped)

#### AmmGnlTC5.var
```iecst
VAR
	iCnt : UINT;
END_VAR
```

### Package Logical/AuxiliariesGeneral - AG: Auxiliaries General

### Data object Logical/AuxiliariesGeneral/META_AG (Simple) - MODUL META data file

#### META_AG.dat
```
; *******************************************************************************
; AGGR: Module Meta Data (data module)
;
; This code is confidential and proprietary to the INNIO Company.
; It may not be used in any form, or reproduced in any manner, without the express
; written permission of the INNIO Company.
; Copyright, INNIO Company, 2025
;
; Customized modifications: -
; ------------------------
;
; History:
; -------
; V03.99.00.00	06.03.2013	Weitzer 	generated for modular software
;			    02.10.2013	lettenb.	descriptions setted
;				04.12.2013				dependencies added
; V04.00.00.00	29.01.2014	lettenb.	1017,1018,1023,1051,3322 UL depended reset 624
; V04.00.01.00	08.05.2014	lettenb.	version changed
; V04.01.00.00	22.05.2014	lettenb.	version changed, interface to GM added
;				01.08.2014	Tinello		OUT_AG.bMsg1120 added
; V04.03.00.00	02.03.2015	lettenb.	version + dependencies changed (920, engine bearing temp. -> MM_EG)
; V04.03.00.00	11.06.2015	Zengerer	version + dependencies changed (IF change with array index 0 for compatibility with c-tasks)
;				15.06.2015  lettenb.	PARAMETER_CHK expanded
; V04.04.00.00	10.05.2016	lettenb.	version + dependencies changed (920)
; V04.04.00.00	12.07.2016	Zengerer 	increase version number for changed customized array size
;               20.03.2017	lettenb.	624: service mode prelubrication added, start delay 6->0s, meas.siganl plaus.check acc. funct.safety
; V04.05.00.00	27.03.2017	lettenb.	BR9: prelubrication for fast start
;				18.07.2017	Messner		Oil circuit fast start V2
;				07.08.2017 	Messner		Starter battery voltage monitoring
;				20.09.2017	Messner		Active Cooling Program added
;				28.07.2017	502423184	due TO SWAT #3: warning added to the oil level minimum
;										due TO SWAT #3: no block OF the pre-heating due TO measuring failure OF oil pan temperatur AND
;										use enigne oil inlet temperature as a fall-back signal FOR the pre-heating
;				19.12.2017	Messner		Oil preheating valve operation messages (B2956, B2957) added
; V04.05.01.00  14.02.2018	Weitzer		EOP_BWS2 added; correction MsgAG, EleStart, AuxGnl after validation
;				28.02.2018	lettenb.	rDPr_BbFilt_A,rDPr_BbFilt_B prepared for vis
; V04.05.02.00  09.04.2018	lettenb.	2770-2784 bParaSetupOk added to avoid alarm at plc startup,bugfix
;               18.09.2018	lettenb.	2233,2432, switch off bat.charger for elestart, bu
; V04.06.00.00  16.07.2018	Perktold	Louvers closed signal added
;										permanent prelube added type 4/6
;				09.10.2018	Schmid		changes in permanent prelube type 4 + type 6 (TC oil valve, W9222+W9225 delayed)
; V04.07.00.00  26.04.2018	lettenb.	SWAT920/5 added
;				09.08.2018	Schmid		2nd low temperature charge cooling circuit added, includes change in tManAuxCtr struct
;				08.01.2019	Schmid		redundant pump control for HWP, CCWP, CC2WP and EmCWP added
;				22.03.2018	Schmid		stop turbo charger cool down run if emergency stop button is pressed, gearbox oil quality sensor removed
; V04.07.01.00	19.06.2019	Schmid		Aux_6: bugfix engine start release from perm. prelube
;										Aux_9: decided on conditions for permanent prelube (30s fast start)/interval prelube (300s fast start)
;				24.06.2019	Schmid		measurement signal failures not restricted by operation mode selector switch (affected W2627, W2628, W2786)
; V04.09.00.00	05.07.2019	Schmidt		added failed TC post-cooling detection/counter
; V04.09.01.00	22.04.2020	Schmid		bugfix in activation of A1017 oil pressure minimum monitoring
; V04.10.00.00	20.07.2020	Schmid		allow fast start without ECWP_Op feedback, failure triggers A1090 during start-up,  W3497 failure in safety loop extended
;				19.11.2020	lettenb.	2348,2349,2350,2351,2352,2353,2355,2359,2360 added
;				03.12.2020	Perktold,	added oil and coolant management
; V04.10.01.00	09.03.2021	Schmid,		bugfix type6 A1060 for IN_AG.bEng_Dem_EPS: min pressure limit for 1 pump instead of 2
;				11.03.2021	lettenb.	9004->9048, Msg# already used, bugfix
; V04.11.00.00	25.11.2021	Schmid		W9279 only active if emergency cooler pump demanded
;				28.01.2022	Perktold	included plant controller upgrade
; V04.11.01.00	04.02.2022	Schmid		oil quality sensor CAN oil configuration for 2nd generation sensor reworked
;				08.02.2022	Schmid		bugfixes control battery check extension
; V04.11.02.00	22.02.2022	Schmid		oil quality sensor modifications from validation + J920 start prelube with auxiliaries demand instead of engine demand
; V04.12.00.00	19.09.2022	Zengerer	new task OilTank for plant oil tank handling
; 				19.12.2022	Perktold	added comments for sr-code (EN 13849-1 / 4.6.3) for W3507
; 				19.12.2022	Perktold	Ctr_ECW, Ctr_EOVal: retrigger caused by X >= WMin just once per controller activation
; 				21.12.2022	Perktold	added W9369 Failure auxiliaries supply voltage engine
;				22.12.2022  Bacci		version changed, starter moitoring improvement, added a delay for starter-charging units batteries reconnection
;				29.03.2023	Tinello		permanent prelubrication with DC pump in case of mains failure / release oil refill set to 10 min / bugfix #1092 oil counter reset
; V04.13.00.00	21.07.2023	Bacci		Type3 new starting procedure and adaptive first start attempt
;				28.07.2023	Tinello		Blow-by fan needs to be operated when oil pump is running (2022-134)
;				03.08.2023	Tinello		BugFix #1236 no engine start in preheating mode
;				27.09.2023	Bacci		Flucon sensor clean-up
;				03.10.2023  Tinello		Bugfix #1266 Heat water pump with softstarter
;				03.10.2023	Tinello		Bugfix #1267 Demand for emergency cooling circuit pump was missing
;				08.11.2023	Tinello		oil refill monitoring, oil level high warning (W2435), bus signal for stopping external EO refill pump (2022-131)
;										ECW pump difference pressure monitoring for all engine types available (2023-185)
;				20.11.2023	Bacci		Starter/s correct engagement monitoring added. A2377, A2378, A2379, B9089, B9090 and B9091 added.
;				07.12.2023 	Tinello		BugFix #918  Consider different types of in- and outlet louvers
;				13.12.2023	Tinello		QC3111 oil pre-heating to avoid high oil pressure at engine start (2023-197)
;				20.12.2023	Tinello		Oil filter diff pressure monitoring (2023-184) - including issue #1122 and Fracas #3216
;				05.03.2024	Bacci		Changes on trip 1120 added
; V4.14.00.00	17.10.2024	Racero		Buffer battery test logic adapted, test runs also during engine operation not only standstill
;				28.10.2024	Nagy		QC2509 Start preparation keeps running issue fix
;				11.11.2024	Zengerer	new task OilFill
;				25.11.2024	Bacci		T6 Start procedure with purge start (2024-219)
;				11.12.2024	Nagy		W9513 Oil refilling failure added, A1043 modified (2024-225)
;				12.12.2024	Nagy		Louvers removed from Auxiliary check and moved to ventillation as a new alarm (2024-226)
;				19.03.2025	Tinello		Issue #1694 Each TC of an overhauled engine, should be able to be cooled with oil
;				08.04.2025	Tinello		SafetyPLC: Deactivated W3497 in case of existing SAFETY-PLC
; V04.25.00.00 	10.07.2025	Tinello	 	SafetyPLC: release for HWP / purge air calculation / Changed behavior of A1053 and A1054 / added gas and fire system failure
;
; Instructions for use:
; --------------------
; make only changes at the version numbers
;
; Outstandings:
; ------------
;
; *******************************************************************************
;
"<META>"
;
; Module ID: 18241
"<MODUL>AG</MODUL>"
;
; Module Version (xx.yy.zz.cc)
"<VERSION>04.25.00.00</VERSION>"
;
; Module Basisupdate Version BU (00-99)
"<BASISUPDATE_VERSION>00</BASISUPDATE_VERSION>"
;
; Optional: specify order number for limitated module usage
"<ORDER></ORDER>" ;<!--(optional for restricted customizations; missing statement makes module valid for all orders)-->
;
; Parameter Check <PARAn Name='aAbcdef' MIN='xxx' MAX='yyy' />  (watch for correct spacings and apostrophs!)
"<PARAMETER_CHK>"
"<PARA1 Name='iEng_Motortype' MIN='208' MAX='920' />"
"<PARA2 Name='rN_EngStart_LimHi' MIN='50.0' MAX='2200.0' />"
"<PARA3 Name='rN_EngNom' MIN='100.0' MAX='2200.0' />"
"<PARA4 Name='tiPreLube' MIN='2000' MAX='300000' />"
"<PARA5 />"
"</PARAMETER_CHK>"
;
; Statement, if engine operation is also allowed without this module (FALSE) or if this module´s parameter check passing is mandatory (TRUE)
"<MANDATORYMODULE>TRUE</MANDATORYMODULE>"
;
; Permanent Datamodule Filenames<!-- NAME ist ohne Dateiendung einzutragen; Nur für Counter und interne Parameter verwenden-->
"<DATAMODULES>" ;<!-- optional; mehrere DATAMODULES erlaubt-->
"	<DATAMODULE>par_AG</DATAMODULE>"
"	<DATAMODULE>oil_perm</DATAMODULE>"
"	<DATAMODULE>perm_AG</DATAMODULE>"
"	<DATAMODULE>OQS_perm</DATAMODULE>"
"</DATAMODULES>"
;
; Dependencies Modules (MMxx.yy.zz.cc)
"<DEPENDENCIES>"
"	<DEPENDENCY MODULE='AB' VERSION='04.00.00.00' />"
"	<DEPENDENCY MODULE='PB' VERSION='04.06.00.00' />"		;new permanent file info
"	<DEPENDENCY MODULE='IG' VERSION='04.13.00.00' />"
"	<DEPENDENCY MODULE='EC' VERSION='04.11.00.00' />"
"	<DEPENDENCY MODULE='EX' VERSION='04.10.00.00' />"
"	<DEPENDENCY MODULE='OP' VERSION='04.14.00.00' />"
"	<DEPENDENCY MODULE='CU' VERSION='04.14.00.00' />"
"	<DEPENDENCY MODULE='GC' VERSION='04.03.00.00' />"
"	<DEPENDENCY MODULE='GM' VERSION='04.01.00.00' />"
"	<DEPENDENCY MODULE='GT' VERSION='04.25.00.00' />"
"	<DEPENDENCY MODULE='EG' VERSION='04.25.00.00' />"
"	<DEPENDENCY MODULE='SY' VERSION='04.00.00.00' />"
"	<DEPENDENCY MODULE='HC' VERSION='04.11.00.00' />"
"	<DEPENDENCY MODULE='HA' VERSION='04.25.00.00' />"
"	<DEPENDENCY MODULE='VE' VERSION='04.14.00.00' />"
"	<DEPENDENCY MODULE='VI' VERSION='04.06.00.00' />"    ; corrected for SW download via HMI
"   <DEPENDENCY VISVERSION='02.15.00.00' />"				;Dependencies Visualization
"</DEPENDENCIES>"
;
; Module function description
"<MODULEFUNCTION>" ;<!-- short overview documentation of module function; add reference to detailed information, if available-->
"	<General>	"
"	Engine auxiliaries control "
"	</General>	"
""
"	<F1 Name='Engine starter' LastModified='4.03.00.00'>"
"	Electrical starter control	"
"	Air starter control	"
"	</F1>"
"	<F2 Name='Engine auxiliaries control' LastModified='4.04.00.00'>"
"	Engine/turbocharger oil pumps, engine water pumps.	"
"	</F2>"
"	<F3 Name='Engine oil counter' LastModified='4.03.00.00'>"
"	Engine oil consumption metering.	"
"	</F3>"
"	<F4 Name='Engine oil condition' LastModified='4.04.00.00'>"
"	Engine oil condition monitoring.	"
"	</F4>"
"	<F5 Name='Engine oil temperature' LastModified='4.02.00.00'>"
"	Engine oil temperature controller. High temperature circuit	"
"	Engine oil temperature controller. Low temperature circuit	"
"	</F5>"
"	<F6 Name='Engine cooling water temperature' LastModified='4.02.00.00'>"
"	Engine cooling water temperature controller.	"
"	</F6>"
"	<F7 Name='Blowby control' LastModified='4.03.00.00'>"
"	Engine crank case pressure controller.	"
"	</F7>"
""
"	<Info>"
" 	UPDATE 4.01.01.00: Perm datamodule moved from SYS- to USERROM	"
"	UPDATE 4.02.01.00: version + dependencies changed (IF change with array index 0 for compatibility with c-tasks)	"
"	UPDATE 4.05.00.00: active cooling added "
"	UPDATE 4.06.00.00: transmit perm status info "
"	UPDATE 4.07.00.00: hydraulic ECW pre-heating (type3+4), redundant pump control "
"	UPDATE 4.14.00.00: new task OilFill prepared "
"	</Info>"
""
"	<Customized LastModified='4.00.00.00'>"
"	- Nothing"
"	</Customized>	"
""
"</MODULEFUNCTION>"
;
"</META>"
```
